PROGRAM MAIN
VAR
;
END_VAR

TrafficLgiht();
Convert();

END_PROGRAM

(* stored: Version 1.1.0.1, ProductVersion 3.1.4024.11
   POU MAIN: Id {86261e5a-b529-4817-93a2-323b76b5469b}, SpecialFunc None *)
